FUNCTION F_BaseplateChillerEnable : BOOL
VAR_INPUT
END_VAR
VAR_IN_OUT CONSTANT
	stErrors : ST_ErrorStates;
END_VAR
VAR
END_VAR

F_BaseplateChillerEnable := FALSE;

IF stErrors.bHardwareFailure THEN
	RETURN;
END_IF

IF stErrors.bLeakUnderTable THEN
	RETURN;
END_IF

F_BaseplateChillerEnable := TRUE;

END_FUNCTION

(* stored: Version 1.1.0.1, ProductVersion 3.1.4020.14
   POU F_BaseplateChillerEnable: Id {1364b9de-d1e4-4cd9-be0a-b8eefa4075df}, SpecialFunc None *)
